(* IEC 61131-3 sources: eCockpitGit/test_project/src/%F%00 Library/%F%Common Functions/%F%Linearsation/%F%DINT TO REAL, 1 file *)

(* ---- %POU%FU_di_r_LinearXEnds.st ---- *)
//This function, converts an x, value to an y value using and x amount of points on the x and y scale
//This function has ends, which means the output is never greater or smaller than the range of y
// |**Version**|**Author**| **Date** |**Changes**
// | 1         | NSN      | 03-01-18 | Creation
FUNCTION FU_di_r_LinearXEnds : REAL
VAR_INPUT
	xIn			:DINT;				//Input value to be linearised
	pXArray		:POINTER TO DINT;	//Address of x array
	pYArray		:POINTER TO REAL; 	//Address of y array
	uiSize		:UINT;				//Amount of points in
END_VAR
VAR
	LowerLimit	:BOOL;
	UpperLimit	:BOOL;
	UpperXAdr	:POINTER TO DINT;	//Buffer for current x address
	LowerXAdr	:POINTER TO DINT;	//Buffer for current x address
	UpperYAdr	:POINTER TO REAL; 	//Buffer for current y address
	LowerYAdr	:POINTER TO REAL; 	//Buffer for current y address
	FOR1		:UINT;
	a			:REAL;
	b			:REAL;
	d			:BOOL;
END_VAR
(*%!%__DELIMITER__%!%*)
IF uiSize > 1 THEN
	//Direction is found
	UpperXAdr					:=		pXArray + 4;
	d							:=		UpperXAdr^ > pXArray^;

	//Pointers are set
	UpperXAdr					:=		pXArray;
	UpperYAdr					:=		pYArray;

	FOR FOR1 := 1 TO uiSize DO
		IF d THEN
			IF UpperXAdr^ <= xIn THEN
				IF FOR1 = uiSize AND UpperXAdr^ <> xIn THEN
					UpperLimit	:=		TRUE;
				ELSIF FOR1 <> uiSize THEN
					UpperXAdr	:=		UpperXAdr + 4;
					UpperYAdr	:=		UpperYAdr + 4;
				END_IF
			ELSE
				IF pXArray = UpperXAdr THEN
					LowerLimit	:=		TRUE;
				ELSE
					LowerXAdr	:=		UpperXAdr - 4;
					LowerYAdr	:=		UpperYAdr - 4;
				END_IF
				Exit;
			END_IF
		ELSE
			IF UpperXAdr^ >= xIn THEN
				IF FOR1 = uiSize AND UpperXAdr^ <> xIn THEN
					UpperLimit	:=		TRUE;
				ELSIF FOR1 <> uiSize THEN
					UpperXAdr	:=		UpperXAdr + 4;
					UpperYAdr	:=		UpperYAdr + 4;
				END_IF
			ELSE
				IF pXArray = UpperXAdr THEN
					LowerLimit	:=		TRUE;
				ELSE
					LowerXAdr	:=		UpperXAdr - 4;
					LowerYAdr	:=		UpperYAdr - 4;
				END_IF
				Exit;
			END_IF
		END_IF
	END_FOR

	IF LowerLimit THEN
		FU_di_r_LinearXEnds			:=		pYArray^;
	ELSIF UpperLimit THEN
		FU_di_r_LinearXEnds			:=		UpperYAdr^;
	ELSE
		IF xIn = UpperXAdr^ THEN
			FU_di_r_LinearXEnds		:=		UpperYAdr^;
		ELSIF xIn = LowerXAdr^ THEN
			FU_di_r_LinearXEnds		:=		LowerYAdr^;
		ELSE
			IF UpperXAdr^ - LowerXAdr^ = 0 THEN
				a					:=		0;
			ELSE
				a					:=		(UpperYAdr^ - LowerYAdr^) / TO_REAL(UpperXAdr^ - LowerXAdr^);
			END_IF
			b						:=		LowerYAdr^ - (a * TO_REAL(LowerXAdr^));
			FU_di_r_LinearXEnds		:=		(a * TO_REAL(xIn)) + b;
		END_IF
	END_IF
END_IF
